// Mitsubishi GX Works2 project: AND   PLC: Q03UDV

PROGRAM MAIN
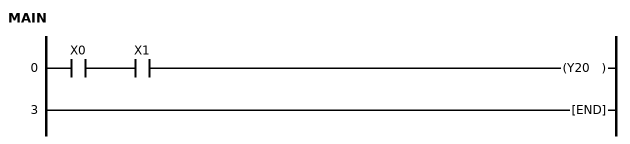
0     LD      X0
      AND     X1
      OUT     Y20
3     END
END_PROGRAM
